FUNCTION F_ComputeUInt32Size : UDINT
VAR_INPUT
    nValue  : UDINT;
END_VAR


F_ComputeUInt32Size := F_ComputeRawVarint32Size(nValue);

END_FUNCTION

(* stored: Version 1.1.0.1
   POU F_ComputeUInt32Size: Id {b832eb68-37ad-415d-ae22-5a35e88c53e7}, SpecialFunc None *)
